PROGRAM MAIN2
VAR
	
	fbSender: FB_MUDPI_SENDER;
	
	{attribute 'OPC.UA.DA' := '0'}
	i_trk_data          AT %I*: PointingKernelPositions;
	
END_VAR



fbSender();
fbSender.SetTimestamp(i_trk_data.time_tai);
fbSender.SetMudpiPayload(ADR(i_trk_data), SIZEOF(i_trk_data));
fbSender.SendData();

END_PROGRAM

(* stored: Version 1.1.0.1, ProductVersion 3.1.4024.9
   POU MAIN2: Id {0130fff6-1a17-435b-ac7d-f0aa5d46a553}, SpecialFunc None *)
